(* Logix 5000 project; controller Lab_4_Traffic_Light_2 vendor 1 type 14 code 150 rev 30.11; software revision 30.00 *)

TASK MainTask (continuous, watchdog 500 ms) : MainProgram

MODULES
   Local : vendor 1 type 14 code 150 (Compact 0, rev 30.11)
      Discrete_IO : Embedded (Compact 1, rev 3.1, Output RPI 20 ms)
      Analog_IO : Embedded (Compact 2, rev 1.1, Output RPI 80 ms)
      Counters : Embedded (Compact 3, rev 1.1, Output RPI 20 ms)
END_MODULES

PROGRAM MainProgram   (* main routine MainRoutine *)
VAR
   ARRAY_1 : DINT[5] := ([1] := 258, [2] := 18, [3] := 513, [4] := 33);
   ARRAY_2 : DINT[5] := ([1] := 4000, [2] := 1000, [3] := 4000, [4] := 1000);
   CONTROL_1 : CONTROL := (LEN := 4, POS := 3);
   CONTROL_2 : CONTROL := (LEN := 4, POS := 3);
   OUTPUT : DINT := 513;
   PV_Green_North : BOOL;
   PV_Green_South : BOOL := 1;
   PV_Red_North : BOOL := 1;
   PV_Red_South : BOOL;
   PV_Yellow_North : BOOL;
   PV_Yellow_South : BOOL;
   T4_1 : TIMER := (PRE := 4000, ACC := 157, EN := 1, TT := 1);   // ON TIMER
END_VAR

ROUTINE MainRoutine   (* ladder *)
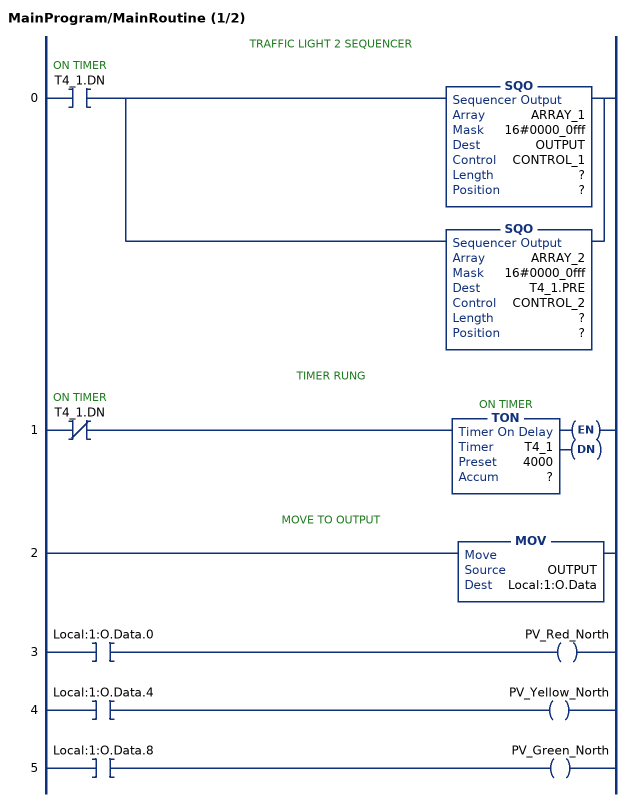
   // TRAFFIC LIGHT 2 SEQUENCER
   0: XIC(T4_1.DN)[SQO(ARRAY_1,16#0000_0fff,OUTPUT,CONTROL_1,?,?) ,SQO(ARRAY_2,16#0000_0fff,T4_1.PRE,CONTROL_2,?,?) ];
   // TIMER RUNG
   1: XIO(T4_1.DN)TON(T4_1,?,?);
   // MOVE TO OUTPUT
   2: MOV(OUTPUT,Local:1:O.Data);
   3: XIC(Local:1:O.Data.0)OTE(PV_Red_North);
   4: XIC(Local:1:O.Data.4)OTE(PV_Yellow_North);
   5: XIC(Local:1:O.Data.8)OTE(PV_Green_North);
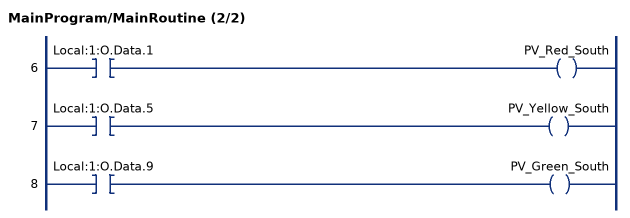
   6: XIC(Local:1:O.Data.1)OTE(PV_Red_South);
   7: XIC(Local:1:O.Data.5)OTE(PV_Yellow_South);
   8: XIC(Local:1:O.Data.9)OTE(PV_Green_South);
END_ROUTINE
END_PROGRAM
